(* CoDeSys 2.3 export: HEATER.EXP *)

(* Global variable list: Heater *)
VAR_GLOBAL

	Heater_AutoSetT_1:					REAL;
	Heater_AutoSetT_2:					REAL;
	Heater_AutoSetT_3:					REAL;
	Heater_AutoSetT_4:					REAL;

END_VAR
